TYPE T_JIG_SOCKET :
STRUCT
	AVAILABLE_SOCKET : ARRAY[0..4] OF DINT;
	LASER_DESTINATION: ARRAY[0..4] OF DINT;
END_STRUCT
END_TYPE

(* stored: Version 1.1.0.1, ProductVersion 3.1.4020.12
   DUT T_JIG_SOCKET: Id {48dab071-1d94-4960-a93e-d7057a9a2c3e} *)
